// TIA Portal V20 export
TYPE "UDT_MTP_ProcedureExtended"
   STRUCT
      Procedure { S7_SetPoint := 'True'} : "UDT_MTP_Procedure";   // Procedure Definition
      StateTransient : Struct   // Transient States
         starting { S7_SetPoint := 'True'} : "UDT_Service_IndexElement";   // Transient State Starting
         running { S7_SetPoint := 'True'} : "UDT_Service_IndexElement";   // Transient State Running
         holding { S7_SetPoint := 'True'} : "UDT_Service_IndexElement";   // Transient State Holding
         unholding { S7_SetPoint := 'True'} : "UDT_Service_IndexElement";   // Transient State Unholding / Transient State Restarting
         pausing { S7_SetPoint := 'True'} : "UDT_Service_IndexElement";   // Transient State Pausing
         resuming { S7_SetPoint := 'True'} : "UDT_Service_IndexElement";   // Transient State Resuming
         completing { S7_SetPoint := 'True'} : "UDT_Service_IndexElement";   // Transient State Completing / Transient State
         stopping { S7_SetPoint := 'True'} : "UDT_Service_IndexElement";   // Transient State stopping / Transient State Stopping / Transient State
         aborting { S7_SetPoint := 'True'} : "UDT_Service_IndexElement";   // Transient State Aborting / Transient State
         resetting { S7_SetPoint := 'True'} : "UDT_Service_IndexElement";   // Transient State Resetting / Transient State
      END_STRUCT;
      ProcedureReportMap : Array[0..0] of DWord;   // Procedure Report Mapping / Procedure Report value Mapping
      ProcedureProcessInMap : Array[0..0] of DWord;   // Procedure Report Mapping / Procedure ProcessIn value Mapping
      ProcedureProcessOutMap : Array[0..0] of DWord;   // Procedure ProcessOut value Mapping
      ProcedureProcedureMap : Array[0..0] of DWord;   // Procedure Procedure parameter Mapping
   END_STRUCT;
END_TYPE
